{attribute 'qualified_only'}
VAR_GLOBAL
    stInputs  : ST_MachineInputs;
    stOutputs : ST_MachineOutputs;
    stCommand : ST_MachineCommand;
    stStatus  : ST_MachineStatus;
    stStationEvents   : ARRAY[0..4] OF ST_StationEvents;
    stEventsAssigment : ST_EventsAssigmentGeneral;
    astActiveEvents   : ARRAY[0..50] OF ST_ActiveEvents;
    sSystemTime       : STRING(255);
    sSystemDate       : STRING(255);
    bMachineFault     : BOOL;
    bCycleStopRequest : BOOL;
END_VAR

(* stored: Version 1.1.0.1, ProductVersion 3.1.4026.18
   GVL GVL_MASTER: Id {9970f182-028c-4164-bcf7-ddc50b57d0ed} *)
